{attribute 'qualified_only'}
{attribute 'strict'}

TYPE ePNcouplerType :
(
	None := 0,
	ModbusTCP:= 1,
	Profinet := 2,
	ModbusTCPV2 := 3
);
END_TYPE

(* stored: Version 1.1.0.1, ProductVersion 3.1.4026.18
   DUT ePNcouplerType: Id {1f6fc4f1-31a7-4712-a708-fb30271525ba} *)
